FUNCTION_BLOCK FB_System_HES_Ablaufsteuerung
VAR_IN_OUT
	Zustand					: ST_System_HES_Zustand;
	Stellwert				: ST_System_HES_Stellwert;
	Steuerung				: ST_System_HES_Steuerung;
END_VAR
VAR_INPUT
	Zustand_Stellventil		: ST_SV_Zustand;
	Zustand_Pumpe			: ST_PU_Zustand;
END_VAR
VAR_OUTPUT
END_VAR
VAR
	E_System_HES_Zustand_Status_Nachl_Stellventil	: SINT;
	E_System_HES_Zustand_Status_Nachl_Pumpe			: SINT;
	E_System_HES_Zustand_Status_Betrieb				: SINT;
	E_System_HES_Zustand_Status_Betrieb_Sperre		: SINT;
	E_System_HES_Zustand_Status_Vorl_Pumpe			: SINT;
	E_System_HES_Zustand_Status_Vorl_Stellventil	: SINT;
	E_System_HES_Zustand_Status_Betriebsbereit		: SINT;
	E_System_HES_Zustand_Status_Stoerung			: SINT;
	E_System_HES_Zustand_Status_Idle_Sperre			: SINT;



END_VAR

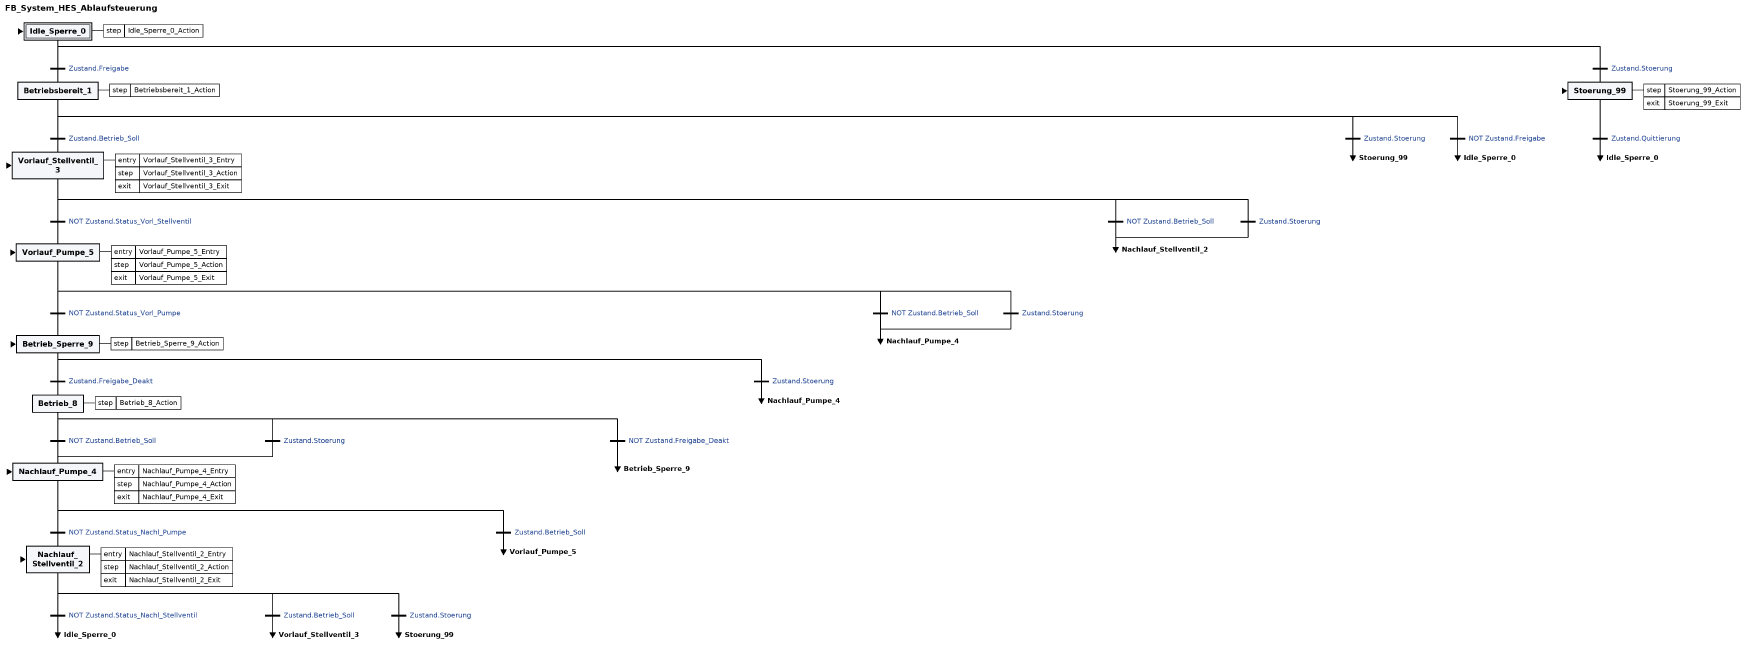
INITIAL_STEP Idle_Sperre_0:
    Idle_Sperre_0_Action(N);  // step action
END_STEP
TRANSITION FROM Idle_Sperre_0 TO Betriebsbereit_1
    := Zustand.Freigabe;
END_TRANSITION
TRANSITION FROM Idle_Sperre_0 TO Stoerung_99
    := Zustand.Stoerung;
END_TRANSITION
STEP Stoerung_99:
    Stoerung_99_Action(N);  // step action
    Stoerung_99_Exit(P0);  // exit action
END_STEP
TRANSITION FROM Stoerung_99 TO Idle_Sperre_0
    := Zustand.Quittierung;
END_TRANSITION
STEP Betriebsbereit_1:
    Betriebsbereit_1_Action(N);  // step action
END_STEP
TRANSITION FROM Betriebsbereit_1 TO Vorlauf_Stellventil_3
    := Zustand.Betrieb_Soll;
END_TRANSITION
TRANSITION FROM Betriebsbereit_1 TO Stoerung_99
    := Zustand.Stoerung;
END_TRANSITION
TRANSITION FROM Betriebsbereit_1 TO Idle_Sperre_0
    := NOT Zustand.Freigabe;
END_TRANSITION
STEP Vorlauf_Stellventil_3:
    Vorlauf_Stellventil_3_Entry(P1);  // entry action
    Vorlauf_Stellventil_3_Action(N);  // step action
    Vorlauf_Stellventil_3_Exit(P0);  // exit action
END_STEP
TRANSITION FROM Vorlauf_Stellventil_3 TO Vorlauf_Pumpe_5
    := NOT Zustand.Status_Vorl_Stellventil;
END_TRANSITION
TRANSITION FROM Vorlauf_Stellventil_3 TO Nachlauf_Stellventil_2
    := NOT Zustand.Betrieb_Soll;
END_TRANSITION
TRANSITION FROM Vorlauf_Stellventil_3 TO Nachlauf_Stellventil_2
    := Zustand.Stoerung;
END_TRANSITION
STEP Vorlauf_Pumpe_5:
    Vorlauf_Pumpe_5_Entry(P1);  // entry action
    Vorlauf_Pumpe_5_Action(N);  // step action
    Vorlauf_Pumpe_5_Exit(P0);  // exit action
END_STEP
TRANSITION FROM Vorlauf_Pumpe_5 TO Betrieb_Sperre_9
    := NOT Zustand.Status_Vorl_Pumpe;
END_TRANSITION
TRANSITION FROM Vorlauf_Pumpe_5 TO Nachlauf_Pumpe_4
    := NOT Zustand.Betrieb_Soll;
END_TRANSITION
TRANSITION FROM Vorlauf_Pumpe_5 TO Nachlauf_Pumpe_4
    := Zustand.Stoerung;
END_TRANSITION
STEP Betrieb_Sperre_9:
    Betrieb_Sperre_9_Action(N);  // step action
END_STEP
TRANSITION FROM Betrieb_Sperre_9 TO Betrieb_8
    := Zustand.Freigabe_Deakt;
END_TRANSITION
TRANSITION FROM Betrieb_Sperre_9 TO Nachlauf_Pumpe_4
    := Zustand.Stoerung;
END_TRANSITION
STEP Betrieb_8:
    Betrieb_8_Action(N);  // step action
END_STEP
TRANSITION FROM Betrieb_8 TO Nachlauf_Pumpe_4
    := NOT Zustand.Betrieb_Soll;
END_TRANSITION
TRANSITION FROM Betrieb_8 TO Nachlauf_Pumpe_4
    := Zustand.Stoerung;
END_TRANSITION
TRANSITION FROM Betrieb_8 TO Betrieb_Sperre_9
    := NOT Zustand.Freigabe_Deakt;
END_TRANSITION
STEP Nachlauf_Pumpe_4:
    Nachlauf_Pumpe_4_Entry(P1);  // entry action
    Nachlauf_Pumpe_4_Action(N);  // step action
    Nachlauf_Pumpe_4_Exit(P0);  // exit action
END_STEP
TRANSITION FROM Nachlauf_Pumpe_4 TO Nachlauf_Stellventil_2
    := NOT Zustand.Status_Nachl_Pumpe;
END_TRANSITION
TRANSITION FROM Nachlauf_Pumpe_4 TO Vorlauf_Pumpe_5
    := Zustand.Betrieb_Soll;
END_TRANSITION
STEP Nachlauf_Stellventil_2:
    Nachlauf_Stellventil_2_Entry(P1);  // entry action
    Nachlauf_Stellventil_2_Action(N);  // step action
    Nachlauf_Stellventil_2_Exit(P0);  // exit action
END_STEP
TRANSITION FROM Nachlauf_Stellventil_2 TO Idle_Sperre_0
    := NOT Zustand.Status_Nachl_Stellventil;
END_TRANSITION
TRANSITION FROM Nachlauf_Stellventil_2 TO Vorlauf_Stellventil_3
    := Zustand.Betrieb_Soll;
END_TRANSITION
TRANSITION FROM Nachlauf_Stellventil_2 TO Stoerung_99
    := Zustand.Stoerung;
END_TRANSITION

ACTION Betrieb_8_Action:
(* Stellwert setzen *)
Stellwert.Anford_Stellventil		:= TRUE;
Stellwert.Anford_Pumpe		:= TRUE;
Stellwert.Anford_Kompressor			:= TRUE;

(* Zustand setzen *)
Zustand.Status				:= E_System_HES_Zustand_Status_Betrieb;
END_ACTION

ACTION Betrieb_Sperre_9_Action:
(* Stellwert setzen *)
Stellwert.Anford_Stellventil		:= TRUE;
Stellwert.Anford_Pumpe		:= TRUE;
Stellwert.Anford_Kompressor			:= TRUE;

(* Zustand setzen *)
Zustand.Status				:= E_System_HES_Zustand_Status_Betrieb_Sperre;
END_ACTION

ACTION Betriebsbereit_1_Action:
(* Stellwert setzen *)
Stellwert.Anford_Stellventil	:= FALSE;
Stellwert.Anford_Pumpe	:= FALSE;
Stellwert.Anford_Kompressor		:= FALSE;

(* Zustand setzen *)
Zustand.Status			:= E_System_HES_Zustand_Status_Betriebsbereit;
END_ACTION

ACTION Idle_Sperre_0_Action:
(* Stellwert setzen *)
Stellwert.Anford_Stellventil	:= FALSE;
Stellwert.Anford_Pumpe			:= FALSE;
Stellwert.Anford_Kompressor		:= FALSE;

(* Zustand setzen *)
Zustand.Status			:= E_System_HES_Zustand_Status_Idle_Sperre;

(* Quittierungszustand auf False setzen, damit das System bei einer erneuten Störung nicht direkt wieder angeschaltet wird *)
Steuerung.Quittierung	:= FALSE;
END_ACTION

ACTION Nachlauf_Pumpe_4_Action:
(* Stellwert setzen *)
Stellwert.Anford_Stellventil		:= TRUE;
Stellwert.Anford_Pumpe		:= FALSE;
Stellwert.Anford_Kompressor			:= FALSE;

(* Zustand setzen *)
Zustand.Status				:= E_System_HES_Zustand_Status_Nachl_Pumpe;
Zustand.Status_Nachl_Pumpe	:= Zustand_Pumpe.Betrieb OR Zustand_Pumpe.Status_Nachl;
END_ACTION

ACTION Nachlauf_Pumpe_4_Entry:
Zustand.Status_Nachl_Pumpe	:= TRUE;
END_ACTION

ACTION Nachlauf_Pumpe_4_Exit:
Zustand.Status_Nachl_Pumpe	:= FALSE;
END_ACTION

ACTION Nachlauf_Stellventil_2_Action:
(* Stellwert setzen *)
Stellwert.Anford_Stellventil		:= FALSE;
Stellwert.Anford_Pumpe		:= FALSE;
Stellwert.Anford_Kompressor			:= FALSE;

(* Zustand setzen *)
Zustand.Status				:= E_System_HES_Zustand_Status_Nachl_Stellventil;
Zustand.Status_Nachl_Stellventil	:= Zustand_Stellventil.Stellung OR Zustand_Stellventil.Stellungwechsel10;
END_ACTION

ACTION Nachlauf_Stellventil_2_Entry:
Zustand.Status_Nachl_Stellventil	:= TRUE;
END_ACTION

ACTION Nachlauf_Stellventil_2_Exit:
Zustand.Status_Nachl_Stellventil	:= FALSE;
END_ACTION

ACTION Stoerung_99_Action:
(* Stellwert setzen *)
Stellwert.Anford_Stellventil	:= FALSE;
Stellwert.Anford_Pumpe	:= FALSE;
Stellwert.Anford_Kompressor		:= FALSE;

(* Zustand setzen *)
Zustand.Stoerung			:= TRUE;
Zustand.Status			:= E_System_HES_Zustand_Status_Stoerung;
END_ACTION

ACTION Stoerung_99_Exit:
Zustand.Stoerung	:= FALSE;
END_ACTION

ACTION Vorlauf_Pumpe_5_Action:
(* Stellwert setzen *)
Stellwert.Anford_Stellventil		:= TRUE;
Stellwert.Anford_Pumpe		:= TRUE;
Stellwert.Anford_Kompressor			:= FALSE;

(* Zustand setzen *)
Zustand.Status				:= E_System_HES_Zustand_Status_Vorl_Pumpe;
Zustand.Status_Vorl_Pumpe	:= NOT(Zustand_Pumpe.Betrieb AND NOT Zustand_Pumpe.Status_Vorl);
END_ACTION

ACTION Vorlauf_Pumpe_5_Entry:
Zustand.Status_Vorl_Pumpe	:= TRUE;
END_ACTION

ACTION Vorlauf_Pumpe_5_Exit:
Zustand.Status_Vorl_Pumpe	:= FALSE;
END_ACTION

ACTION Vorlauf_Stellventil_3_Action:
(* Stellwert setzen *)
Stellwert.Anford_Stellventil		:= TRUE;
Stellwert.Anford_Pumpe		:= FALSE;
Stellwert.Anford_Kompressor			:= FALSE;

(* Zustand setzen *)
Zustand.Status				:= E_System_HES_Zustand_Status_Vorl_Stellventil;
Zustand.Status_Vorl_Stellventil	:= NOT(Zustand_Stellventil.Stellung AND NOT Zustand_Stellventil.Stellungwechsel01);
END_ACTION

ACTION Vorlauf_Stellventil_3_Entry:
Zustand.Status_Vorl_Stellventil	:= TRUE;
END_ACTION

ACTION Vorlauf_Stellventil_3_Exit:
Zustand.Status_Vorl_Stellventil	:= FALSE;
END_ACTION

END_FUNCTION_BLOCK

(* stored: Version 1.1.0.1, ProductVersion 3.1.4024.9
   POU FB_System_HES_Ablaufsteuerung: Id {846c77d2-353c-49c0-ae9b-98e2051d871e}, SpecialFunc None
   Action Betrieb_8_Action: Id {5070df7f-508d-4f1d-af6e-689b6393d3ae}
   Action Betrieb_Sperre_9_Action: Id {bf5d54ee-bcb1-4d6c-a87f-0616d2830ff1}
   Action Betriebsbereit_1_Action: Id {4d6a1016-fb55-4528-a712-5c06bea7a279}
   Action Idle_Sperre_0_Action: Id {bbd32a28-31ff-4760-acf7-ddc7d4af48a3}
   Action Nachlauf_Pumpe_4_Action: Id {f0fceb22-37b6-42bd-a28f-ccf7096c3c23}
   Action Nachlauf_Pumpe_4_Entry: Id {4fdf4178-19b1-41b2-8460-b485b2ad405f}
   Action Nachlauf_Pumpe_4_Exit: Id {b291d98a-2784-4a6a-bf7b-eda0f29cf67b}
   Action Nachlauf_Stellventil_2_Action: Id {81e2f1ee-3a95-4164-94bf-6d1905c7a1d1}
   Action Nachlauf_Stellventil_2_Entry: Id {25180ecb-35bb-4ca6-9aeb-0435582e3d9a}
   Action Nachlauf_Stellventil_2_Exit: Id {5ad8ae12-60be-40d1-82b7-d41617d782b0}
   Action Stoerung_99_Action: Id {354e8881-f624-4843-b97d-a59b7066a5e0}
   Action Stoerung_99_Exit: Id {ef80a896-6768-4205-bf1e-b24afe4d3a53}
   Action Vorlauf_Pumpe_5_Action: Id {69a94baa-9617-4266-a42b-200e1561a462}
   Action Vorlauf_Pumpe_5_Entry: Id {0c0cb81f-b194-48d3-9ca5-bc3cd8062be7}
   Action Vorlauf_Pumpe_5_Exit: Id {5114be12-f8ce-4a78-b141-86a9dd23e4c2}
   Action Vorlauf_Stellventil_3_Action: Id {e3ead50b-85a8-4b5a-99df-eb4039b0cf85}
   Action Vorlauf_Stellventil_3_Entry: Id {d20a5fa1-cdc4-42fb-a060-011d99358219}
   Action Vorlauf_Stellventil_3_Exit: Id {ebc6a50d-2b65-48a2-9361-d39c342c4f1e} *)
